PROGRAM MAIN
VAR
END_VAR

END_PROGRAM

(* stored: Version 1.1.0.1
   POU MAIN: Id {4679dd22-b08c-42f7-9135-68ffa896d139} *)
